// TIA Portal V20 export
DATA_BLOCK "BK31"   // DB279
// stored: MemoryReserve 100
   VAR
      "ANODE MAIN P&P1 VACUUM ON" : Bool := FALSE;
      "ANODE MAIN P&P1 VACUUM OFF" : Bool := FALSE;
      "ANODE MAIN P&P2 VACUUM ON" : Bool := FALSE;
      "ANODE MAIN P&P2 VACUUM OFF" : Bool := FALSE;
      "ANODE MAIN NG P&P VACUUM ON" : Bool := FALSE;
      "ANODE MAIN NG P&P VACUUM OFF" : Bool := FALSE;
      "ANODE ALIGN TABLE VACUUM ON" : Bool := FALSE;
      "ANODE ALIGN TABLE VACUUM OFF" : Bool := FALSE;
   END_VAR
BEGIN
END_DATA_BLOCK
